(* IEC 61131-3 sources: plc_generation_empirical_study/datasets/task_bank_c06_reverse_bounded_runtime_v0_3/tasks/C06_V20_lean_composite/negative_control, 1 file *)

(* ---- NC1.st ---- *)
FUNCTION_BLOCK C06_V20_lean_composite
VAR_INPUT
    A_AutoMode : BOOL;
    A_AutoDemand : BOOL;
    A_ManualDemand : BOOL;
    A_SafetyOK : BOOL;
    A_Inhibit : BOOL;
    B_ItemPulse : BOOL;
    B_Rejected : BOOL;
    B_Stop : BOOL;
    B_Reset : BOOL;
    B_Target : INT;
    B_RejectLimit : INT;
    SubsystemBEnable : BOOL;
    CrossReset : BOOL;
END_VAR
VAR_OUTPUT
    A_Command : BOOL;
    A_Blocked : BOOL;
    B_AcceptedCount : INT;
    B_RejectCount : INT;
    B_ConsecutiveRejects : INT;
    B_Complete : BOOL;
    B_LockedOut : BOOL;
    CrossReady : BOOL;
    CrossBlocked : BOOL;
END_VAR
VAR
    B_PrevItem : BOOL;
END_VAR

A_Command := ((A_AutoMode AND A_AutoDemand) OR ((NOT A_AutoMode) AND A_ManualDemand))
           AND A_SafetyOK AND (NOT A_Inhibit);
A_Blocked := ((A_AutoMode AND A_AutoDemand) OR ((NOT A_AutoMode) AND A_ManualDemand))
           AND ((NOT A_SafetyOK) OR A_Inhibit);

IF CrossReset THEN
    CrossReady := FALSE;
ELSIF A_Command THEN
    CrossReady := TRUE;
END_IF;
CrossBlocked := FALSE;

IF SubsystemBEnable AND CrossReady THEN
    IF B_Reset AND B_Stop AND (NOT B_ItemPulse) THEN
        B_AcceptedCount := 0;
        B_RejectCount := 0;
        B_ConsecutiveRejects := 0;
        B_Complete := FALSE;
        B_LockedOut := FALSE;
    ELSIF B_RejectLimit <= 0 THEN
        B_LockedOut := TRUE;
    ELSIF B_ItemPulse AND (NOT B_PrevItem) AND (NOT B_Stop) AND (NOT B_Complete) AND (NOT B_LockedOut) THEN
        IF B_Rejected THEN
            B_RejectCount := B_RejectCount + 1;
            B_ConsecutiveRejects := B_ConsecutiveRejects + 1;
            IF B_ConsecutiveRejects >= B_RejectLimit THEN B_LockedOut := TRUE; END_IF;
        ELSE
            B_AcceptedCount := B_AcceptedCount + 1;
            B_ConsecutiveRejects := 0;
            IF (B_Target > 0) AND (B_AcceptedCount >= B_Target) THEN B_Complete := TRUE; END_IF;
        END_IF;
    END_IF;
    B_PrevItem := B_ItemPulse;
ELSE
    B_AcceptedCount := 0;
    B_RejectCount := 0;
    B_ConsecutiveRejects := 0;
    B_Complete := FALSE;
    B_LockedOut := FALSE;
END_IF;

END_FUNCTION_BLOCK
